// Mitsubishi GX Works2 project: z04   PLC: Q02/Q02H

PROGRAM MAIN
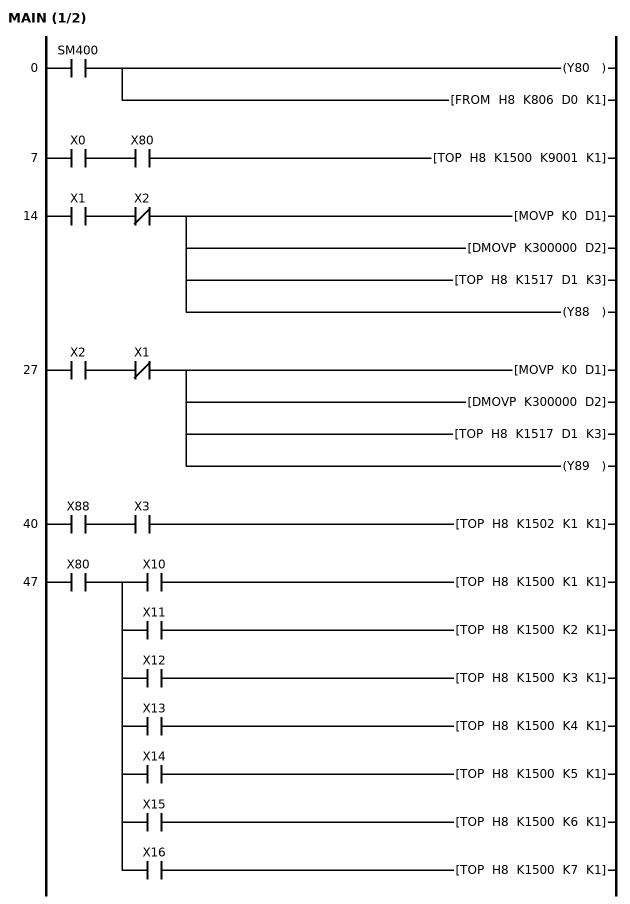
0     LD      SM400
      OUT     Y80
      FROM    H8 K806 D0 K1
7     LD      X0
      AND     X80
      TOP     H8 K1500 K9001 K1
14    LD      X1
      ANI     X2
      MOVP    K0 D1
      DMOVP   K300000 D2
      TOP     H8 K1517 D1 K3
      OUT     Y88
27    LD      X2
      ANI     X1
      MOVP    K0 D1
      DMOVP   K300000 D2
      TOP     H8 K1517 D1 K3
      OUT     Y89
40    LD      X88
      AND     X3
      TOP     H8 K1502 K1 K1
47    LD      X80
      MPS
      AND     X10
      TOP     H8 K1500 K1 K1
      MRD
      AND     X11
      TOP     H8 K1500 K2 K1
      MRD
      AND     X12
      TOP     H8 K1500 K3 K1
      MRD
      AND     X13
      TOP     H8 K1500 K4 K1
      MRD
      AND     X14
      TOP     H8 K1500 K5 K1
      MRD
      AND     X15
      TOP     H8 K1500 K6 K1
      MPP
      AND     X16
      TOP     H8 K1500 K7 K1
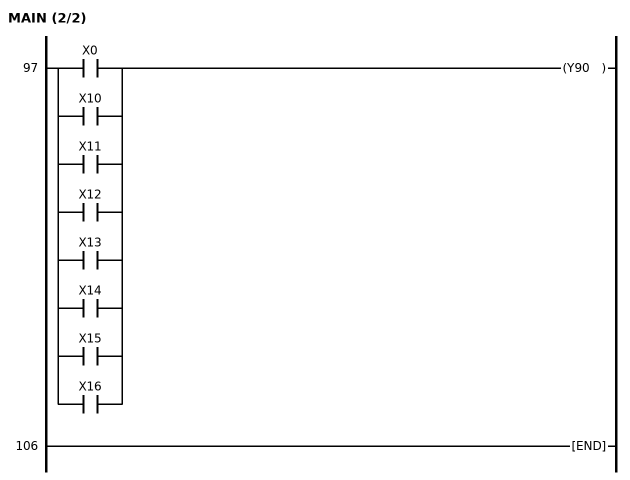
97    LD      X0
      OR      X10
      OR      X11
      OR      X12
      OR      X13
      OR      X14
      OR      X15
      OR      X16
      OUT     Y90
106   END
END_PROGRAM
